// TwinCAT 3 PLC project SILO_OOP_PLC
// ProgramVersion: 3.1.4024.0
// libraries:
//   Tc2_Standard, * (Beckhoff Automation GmbH)
//   Tc2_System, * (Beckhoff Automation GmbH)
//   Tc3_Module, * (Beckhoff Automation GmbH)
// project tree:
//   / PlcTask.TcTTO
//   POUs/1. Interfaces/ itfActuate.TcIO, itfAutoManual.TcIO, itfDetect.TcIO, itfFault.TcIO, itfRamp.TcIO, itfReturnBOOL.TcIO, itfScale.TcIO, itfSiloFlags.TcIO, itfState.TcIO, itfStatusFlags.TcIO
//   POUs/2. Features/ itfActuateImplement.TcPOU, itfFaultImplement.TcPOU, itfRampImplement.TcPOU, itfScaleAnalogInputImplement.TcPOU, itfScaleAnalogOutputImplement.TcPOU, itfDetectImplement.TcPOU, itfSiloFlagsImplement.TcPOU, itfStatusFlagsImplement.TcPOU
//   POUs/3. IO Structure/ GateI.TcDUT, GateO.TcDUT, LoadCellI.TcDUT, LoadCellO.TcDUT, MotorI.TcDUT, MotorO.TcDUT, ProxI.TcDUT, VFDI.TcDUT, VFDO.TcDUT
//   POUs/4. Actuators/ Gate.TcPOU, Motor.TcPOU, VFD.TcPOU
//   POUs/5. Sensors/ LoadCell.TcPOU, ProximitySensor.TcPOU
//   POUs/6.Wrapper/ Wrapper.TcPOU
//   POUs/7.FSM/ BaseState.TcPOU, BufferingProduct.TcPOU, ConveyProduct.TcPOU, Dose.TcPOU, DoseInit.TcPOU, GateHandler.TcPOU, MixerDepositCheck.TcPOU, Mixing.TcPOU, NewBatch.TcPOU, StorageCheck.TcPOU
//   POUs/ MAIN.TcPOU
// real-time tasks:
//   TASK PlcTask: cycle T#10ms, priority 20, ADS port 350

CONFIGURATION SILO_OOP_PLC
    RESOURCE PLC ON TwinCAT3
        TASK PlcTask(INTERVAL := T#10ms, PRIORITY := 20);
        PROGRAM MAIN WITH PlcTask : MAIN;
    END_RESOURCE
END_CONFIGURATION

// ---- POUs/3. IO Structure/GateI.TcDUT
TYPE GateI :
STRUCT
	Open : BOOL;
	Close : BOOL;
END_STRUCT
END_TYPE

// ---- POUs/3. IO Structure/GateO.TcDUT
TYPE GateO :
STRUCT
	Coil : BOOL;
END_STRUCT
END_TYPE

// ---- POUs/3. IO Structure/LoadCellI.TcDUT
TYPE LoadCellI :
STRUCT
	AnalogSignal : INT;
	MaxSignalValue : INT;
	MaxUnitValue : INT;
END_STRUCT
END_TYPE

// ---- POUs/3. IO Structure/LoadCellO.TcDUT
TYPE LoadCellO :
STRUCT
	ScaledValue : INT;
END_STRUCT
END_TYPE

// ---- POUs/3. IO Structure/MotorI.TcDUT
TYPE MotorI :
STRUCT
	Start : BOOL;
	Stop : BOOL;
	Overload : BOOL;
	ResetOverload: BOOL;
END_STRUCT
END_TYPE

// ---- POUs/3. IO Structure/MotorO.TcDUT
TYPE MotorO :
STRUCT
	Coil : BOOL;
	FaultStatus : BOOL;
END_STRUCT
END_TYPE

// ---- POUs/3. IO Structure/ProxI.TcDUT
TYPE ProxI :
STRUCT
	Signal : BOOL;
END_STRUCT
END_TYPE

// ---- POUs/3. IO Structure/VFDI.TcDUT
TYPE VFDI EXTENDS MotorI :
STRUCT
	InputFreq : INT;
	RampRate : INT;
	FreqMaxSignal : INT;
END_STRUCT
END_TYPE

// ---- POUs/3. IO Structure/VFDO.TcDUT
TYPE VFDO EXTENDS MotorO :
STRUCT
	OutputFreq : INT;
END_STRUCT
END_TYPE

// ---- POUs/1. Interfaces/itfActuate.TcIO
INTERFACE itfActuate

METHOD mTurnOffAuto : BOOL
VAR_INPUT
END_VAR
END_METHOD

METHOD mTurnOffManual : BOOL
VAR_INPUT
END_VAR
END_METHOD

METHOD mTurnOnAuto : BOOL
VAR_INPUT
END_VAR
END_METHOD

METHOD mTurnOnManual : BOOL
VAR_INPUT
END_VAR
END_METHOD

PROPERTY pCoil : Bool
GET
END_GET
SET
END_SET
END_PROPERTY

PROPERTY pStart : Bool
GET
END_GET
SET
END_SET
END_PROPERTY

PROPERTY pStop : Bool
GET
END_GET
SET
END_SET
END_PROPERTY

END_INTERFACE

// ---- POUs/1. Interfaces/itfAutoManual.TcIO
INTERFACE itfAutoManual

METHOD mAutoOff : BOOL
VAR_INPUT
END_VAR
END_METHOD

METHOD mAutoOn : BOOL
VAR_INPUT
END_VAR
END_METHOD

METHOD mFault : BOOL
VAR_INPUT
END_VAR
END_METHOD

METHOD mManual : BOOL
VAR_INPUT
END_VAR
END_METHOD

METHOD mRunning : BOOL
VAR_INPUT
END_VAR
END_METHOD

END_INTERFACE

// ---- POUs/1. Interfaces/itfDetect.TcIO
INTERFACE itfDetect

PROPERTY pDetectSignal : BOOL
GET
END_GET
SET
END_SET
END_PROPERTY

END_INTERFACE

// ---- POUs/1. Interfaces/itfFault.TcIO
INTERFACE itfFault

METHOD mResetFault : BOOL
VAR_INPUT
END_VAR
END_METHOD

METHOD mSetFault : BOOL
VAR_INPUT
END_VAR
END_METHOD

PROPERTY pFault : Bool
GET
END_GET
SET
END_SET
END_PROPERTY

PROPERTY pFaultStatus : Bool
GET
END_GET
SET
END_SET
END_PROPERTY

PROPERTY pResetButton : BOOL
GET
END_GET
SET
END_SET
END_PROPERTY

END_INTERFACE

// ---- POUs/1. Interfaces/itfRamp.TcIO
INTERFACE itfRamp

METHOD mDoneTargetFreq : BOOL
VAR_INPUT
END_VAR
END_METHOD

METHOD mRampDown : INT
VAR_INPUT
END_VAR
END_METHOD

METHOD mRampUp : INT
VAR_INPUT
END_VAR
END_METHOD

METHOD mTimerScale : INT
VAR_INPUT
END_VAR
END_METHOD

PROPERTY pOutputValue : INT
GET
END_GET
SET
END_SET
END_PROPERTY

PROPERTY pPulsePeriod : INT
GET
END_GET
SET
END_SET
END_PROPERTY

PROPERTY pRampDone : BOOL
GET
END_GET
SET
END_SET
END_PROPERTY

PROPERTY pRampRate : INT
GET
END_GET
SET
END_SET
END_PROPERTY

PROPERTY pTargetFreq : INT
GET
END_GET
SET
END_SET
END_PROPERTY

END_INTERFACE

// ---- POUs/1. Interfaces/itfReturnBOOL.TcIO
INTERFACE itfReturnBOOL

METHOD mReturnBOOL : BOOL
VAR_INPUT
END_VAR
END_METHOD

END_INTERFACE

// ---- POUs/1. Interfaces/itfScale.TcIO
INTERFACE itfScale

METHOD mScale : INT
VAR_INPUT
END_VAR
END_METHOD

PROPERTY pAnalogSignal : INT
GET
END_GET
SET
END_SET
END_PROPERTY

PROPERTY pMaxSignalValue : INT
GET
END_GET
SET
END_SET
END_PROPERTY

PROPERTY pMaxUnitValue : INT
GET
END_GET
SET
END_SET
END_PROPERTY

PROPERTY pScaledSignal : INT
GET
END_GET
SET
END_SET
END_PROPERTY

END_INTERFACE

// ---- POUs/1. Interfaces/itfSiloFlags.TcIO
INTERFACE itfSiloFlags

PROPERTY pBufferedWeight : INT
GET
END_GET
SET
END_SET
END_PROPERTY

PROPERTY pLowProduct : BOOL
GET
END_GET
SET
END_SET
END_PROPERTY

PROPERTY pTargetWeight : INT
GET
END_GET
SET
END_SET
END_PROPERTY

END_INTERFACE

// ---- POUs/1. Interfaces/itfState.TcIO
INTERFACE itfState

METHOD mIrun : BOOL
VAR_INPUT
END_VAR
END_METHOD

END_INTERFACE

// ---- POUs/1. Interfaces/itfStatusFlags.TcIO
INTERFACE itfStatusFlags

PROPERTY pBuffering : BOOL
GET
END_GET
SET
END_SET
END_PROPERTY

PROPERTY pDosing : BOOL
GET
END_GET
SET
END_SET
END_PROPERTY

PROPERTY pFault : BOOL
GET
END_GET
SET
END_SET
END_PROPERTY

PROPERTY pHaltBatch : BOOL
GET
END_GET
SET
END_SET
END_PROPERTY

PROPERTY pLowProduct : BOOL
GET
END_GET
SET
END_SET
END_PROPERTY

PROPERTY pMixing : BOOL
GET
END_GET
SET
END_SET
END_PROPERTY

PROPERTY pStoring : BOOL
GET
END_GET
SET
END_SET
END_PROPERTY

END_INTERFACE

// ---- POUs/MAIN.TcPOU
PROGRAM MAIN
VAR
	Machine1: Wrapper;
	SpiralInput: ARRAY [1..NUM_SILOS] OF VFDI := [(InputFreq := 50, RampRate := 15, FreqMaxSignal := 200), (InputFreq := 45, RampRate := 20, FreqMaxSignal := 200)];
	LoadCellInput: ARRAY [1..NUM_SILOS] OF LoadCellI := [(AnalogSignal := 4000, MaxSignalValue := 10000, MaxUnitValue := 5000), (AnalogSignal := 3000, MaxSignalValue := 10000, MaxUnitValue := 5000)];
	ConveyorInput: ARRAY [1..NUM_CONVEYORS] OF MotorI;
	ElevatorInput: ARRAY [1..NUM_ELEVATORS] OF MotorI;
	MixerInput: ARRAY [1..NUM_MIXERS] OF VFDI;
	GateInput: ARRAY [1..NUM_GATES] OF GateI;
	ProximityInput: ARRAY [1..NUM_PROXIMITY] OF ProxI;
	SpiralOutput: ARRAY [1..NUM_SILOS] OF VFDO;
	LoadCellOutput: ARRAY [1..NUM_SILOS] OF LoadCellO;
	ConveyorOutput: ARRAY [1..NUM_CONVEYORS] OF MotorO;
	ElevatorOutput: ARRAY [1..NUM_ELEVATORS] OF MotorO;
	MixerOutput: ARRAY [1..NUM_MIXERS] OF VFDO;
	GateOutput: ARRAY [1..NUM_GATES] OF GateO;
	
	Buffering : BOOL;
	Dosing : BOOL;
	Fault : BOOL;
	HaltBatch : BOOL;
	Mixing : BOOL;
	Sorting : BOOL;
	
END_VAR
VAR CONSTANT
	NUM_SILOS : INT:=2;
	NUM_GATES : INT:=2;
	NUM_CONVEYORS : INT:=1;
	NUM_ELEVATORS : INT:=1;
	NUM_PROXIMITY : INT:=4;
	NUM_MIXERS : INT:=1;
END_VAR

Machine1(
	SpiralInput:= SpiralInput , 
	LoadCellInput:= LoadCellInput, 
	ConveyorInput:= ConveyorInput, 
	ElevatorInput:= ElevatorInput, 
	MixerInput:= MixerInput, 
	GateInput:= GateInput, 
	ProximityInput:= ProximityInput, 
	SpiralOutput=> SpiralOutput, 
	LoadCellOutput=> LoadCellOutput, 
	ConveyorOutput=> ConveyorOutput, 
	ElevatorOutput=> ElevatorOutput, 
	MixerOutput=> MixerOutput, 
	GateOutput=> GateOutput);

Machine1.SiloFlagsAccessI[1].pTargetWeight := 50;
Machine1.SiloFlagsAccessI[2].pTargetWeight := 80;
	
Buffering := Machine1.MachineFlagsAccessI.pBuffering;
Dosing := Machine1.MachineFlagsAccessI.pDosing;
Fault := Machine1.MachineFlagsAccessI.pFault;
HaltBatch := Machine1.MachineFlagsAccessI.pHaltBatch;
Mixing := Machine1.MachineFlagsAccessI.pMixing;
Sorting := Machine1.MachineFlagsAccessI.pStoring;

END_PROGRAM

// ---- POUs/6.Wrapper/Wrapper.TcPOU
FUNCTION_BLOCK Wrapper
VAR_INPUT
	SpiralInput : ARRAY [1..NUM_SILOS] OF VFDI;
	LoadCellInput : ARRAY [1..NUM_SILOS] OF LoadCellI;
	ConveyorInput : ARRAY [1..NUM_CONVEYORS] OF MotorI;
	ElevatorInput : ARRAY [1..NUM_ELEVATORS] OF MotorI;
	MixerInput : ARRAY [1..NUM_MIXERS] OF VFDI;
	GateInput : ARRAY [1..NUM_GATES] OF GateI;
	ProximityInput : ARRAY [1..NUM_PROXIMITY] OF ProxI;
	
	SpiralAccessI : ARRAY [1..NUM_SILOS] OF itfAutoManual;
	ConveyorAccessI : ARRAY [1..NUM_CONVEYORS] OF itfAutoManual;
	ElevatorAccessI : ARRAY [1..NUM_ELEVATORS] OF itfAutoManual;
	MixerAccessI : ARRAY [1..NUM_MIXERS] OF itfAutoManual;
	GateAccessI : ARRAY [1..NUM_GATES] OF itfAutoManual;
	ProximityAccessI : ARRAY [1..NUM_PROXIMITY] OF itfReturnBOOL;
	MachineFlagsAccessI : itfStatusFlags;
	SiloFlagsAccessI : ARRAY [1..NUM_SILOS] OF itfSiloFlags;
	
	SuperActuator : ARRAY [1..NUM_ACTUATORS] OF itfAutoManual;	
END_VAR
VAR_OUTPUT
	SpiralOutput : ARRAY [1..NUM_SILOS] OF VFDO;
	LoadCellOutput : ARRAY [1..NUM_SILOS] OF LoadCellO;
	ConveyorOutput : ARRAY [1..NUM_CONVEYORS] OF MotorO;
	ElevatorOutput : ARRAY [1..NUM_ELEVATORS] OF MotorO;
	MixerOutput : ARRAY [1..NUM_MIXERS] OF VFDO;
	GateOutput : ARRAY [1..NUM_GATES] OF GateO;
END_VAR
VAR

////////////////////////////////////Actuators//////////////////////////////////////////
	Spiral : ARRAY [0..NUM_SILOS] OF VFD;
	Conveyor : ARRAY [0..NUM_CONVEYORS] OF Motor;
	Elevator : ARRAY [0..NUM_ELEVATORS] OF Motor;
	Mixer : ARRAY [0..NUM_MIXERS] OF VFD;
	Gate : ARRAY [0..NUM_SILOS] OF Gate;
////////////////////////////////////Sensors////////////////////////////////////////////
	LoadCell : ARRAY [0..NUM_SILOS] OF LoadCell;
	Proximities : ARRAY [0..NUM_PROXIMITY] OF ProximitySensor;
///////////////////////////////Machine Flags///////////////////////////////////////////
	MachineFlags : itfStatusFlagsImplement;	
	SiloFlags : ARRAY [0..NUM_SILOS] OF itfSiloFlagsImplement;
	
	INDEX : INT;
	StateIndex : INT := 1;
	IndependentStateIndex : INT :=1;
//////////////////////////////////FSM///////////////////////////////////////////////////
	Execute : ARRAY [1..NUM_STATES] OF itfState;
	Execute_Independent : ARRAY [1..NUM_INDEPENDENT_STATES] OF itfState;
	
	Buffer : BufferingProduct(THIS);
	Convey : ConveyProduct(THIS);
	DoseInitialize : DoseInit(THIS);
	DoseBegin : Dose(THIS);
	Mix : Mixing (THIS);
	GateActuate : GateHandler(THIS);
	Guard : NewBatch(THIS);
	Store : StorageCheck(THIS);
	MixerCheck : MixerDepositCheck(THIS);
//////////////////////////////Fault Handling//////////////////////////////////////////////
	LastStatus : ARRAY[1..NUM_ACTUATORS] OF BOOL;
	
	FaultR : R_TRIG;
	FaultF : F_TRIG;
	
END_VAR
VAR CONSTANT
	NUM_SILOS : INT:=2;
	NUM_GATES : INT:=2;
	NUM_CONVEYORS : INT:=1;
	NUM_ELEVATORS : INT:=1;
	NUM_PROXIMITY : INT:=4;
	NUM_MIXERS : INT:=1;
	
	NUM_ACTUATORS : INT:=7;
	
	NUM_STATES : INT:=9;
	NUM_INDEPENDENT_STATES : INT:=1;
END_VAR

Map();
mManualMode();
StatesMap();

FaultR(CLK:=mCheckFaults());
FaultF(CLK:=mCheckFaults());

IF FaultR.Q THEN
	mSaveActuatorsStatus();
	mGeneralShutDown();
END_IF

IF FaultF.Q THEN
	mRestoreStatus();
END_IF

IF mCheckFaults()=FALSE THEN
	IF pStateIndex > NUM_STATES THEN
		pStateIndex := 1;
	ELSE
		Execute[pStateIndex].mIrun();
	END_IF
	
	Execute_Independent[pIndependentStateIndex].mIrun();
END_IF

METHOD PRIVATE Map : BOOL
VAR_INPUT
END_VAR
FOR INDEX:=1 TO NUM_SILOS BY 1 DO
	SpiralAccessI[INDEX] := Spiral[INDEX];
	Spiral[INDEX](VFDInput:= SpiralInput[INDEX], VFDOutput=>SpiralOutput[INDEX]);
	
	LoadCell[INDEX](LoadCellInput := LoadCellInput[INDEX], LoadCellOutput => LoadCellOutput[INDEX]);

	SiloFlagsAccessI[INDEX] := SiloFlags[INDEX];
END_FOR

FOR INDEX:=1 TO NUM_CONVEYORS BY 1 DO
	ConveyorAccessI[INDEX] := Conveyor[INDEX];
	Conveyor[INDEX](MotorInput:=ConveyorInput[INDEX], MotorOutput=>ConveyorOutput[INDEX]);
END_FOR

FOR INDEX:=1 TO NUM_ELEVATORS BY 1 DO
	ElevatorAccessI[INDEX] := Elevator[INDEX];
	Elevator[INDEX](MotorInput:=ElevatorInput[INDEX], MotorOutput=>ElevatorOutput[INDEX]);
END_FOR

FOR INDEX:=1 TO NUM_MIXERS BY 1 DO
	MixerAccessI[INDEX] := Mixer[INDEX];
	Mixer[INDEX](VFDInput:=MixerInput[INDEX], VFDOutput=>MixerOutput[INDEX]);
END_FOR

FOR INDEX:=1 TO NUM_GATES BY 1 DO
	Gate[INDEX](GateInput:=GateInput[INDEX], GateOutput=>GateOutput[INDEX]);
	GateAccessI[INDEX] := Gate[INDEX];
END_FOR

FOR INDEX:=1 TO NUM_PROXIMITY BY 1 DO
	Proximities[INDEX](ProximityInput:=ProximityInput[INDEX]);
	ProximityAccessI[INDEX] := Proximities[INDEX];
END_FOR

MachineFlagsAccessI := MachineFlags;

SuperActuator[1] := SpiralAccessI[1];
SuperActuator[2] := SpiralAccessI[2];
SuperActuator[3] := ConveyorAccessI[1];
SuperActuator[4] := ElevatorAccessI[1];
SuperActuator[5] := MixerAccessI[1];
SuperActuator[6] := GateAccessI[1];
SuperActuator[7] := GateAccessI[2];
END_METHOD

METHOD PRIVATE mCheckFaults : BOOL
VAR_INPUT
END_VAR
FOR INDEX:=1 TO NUM_ACTUATORS BY 1 DO
	IF SuperActuator[INDEX].mFault() THEN
	THIS^.MachineFlagsAccessI.pFault:=TRUE;
	mCheckFaults:=TRUE;
	RETURN;
END_IF	
END_FOR

MachineFlagsAccessI.pFault:=FALSE;
mCheckFaults:=FALSE;
END_METHOD

METHOD PRIVATE mGeneralShutDown : BOOL
VAR_INPUT
END_VAR
FOR INDEX:=1 TO NUM_ACTUATORS BY 1 DO
	SuperActuator[INDEX].mAutoOff();
END_FOR
END_METHOD

METHOD PRIVATE mManualMode : BOOL
VAR_INPUT
END_VAR
FOR INDEX:=1 TO NUM_ACTUATORS BY 1 DO
	SuperActuator[INDEX].mManual();	
END_FOR
END_METHOD

METHOD PRIVATE mRestoreStatus : BOOL
VAR_INPUT
END_VAR
FOR INDEX:=1 TO NUM_ACTUATORS BY 1 DO
	IF LastStatus[INDEX] = TRUE THEN
		SuperActuator[INDEX].mAutoOn();
	END_IF
END_FOR
END_METHOD

METHOD PRIVATE mSaveActuatorsStatus : BOOL
VAR_INPUT
END_VAR
FOR INDEX:=1 TO NUM_ACTUATORS BY 1 DO
	LastStatus[INDEX]:=SuperActuator[INDEX].mRunning();
END_FOR
END_METHOD

PROPERTY pIndependentStateIndex : INT
GET
pIndependentStateIndex := IndependentStateIndex;
END_GET
SET
IndependentStateIndex := pIndependentStateIndex;
END_SET
END_PROPERTY

PROPERTY pNUM_SILOS : INT
GET
pNUM_SILOS := NUM_SILOS;
END_GET
END_PROPERTY

PROPERTY pStateIndex : INT
GET
pStateIndex := StateIndex;
END_GET
SET
StateIndex := pStateIndex;
END_SET
END_PROPERTY

METHOD PRIVATE StatesMap : BOOL
VAR_INPUT
END_VAR
Execute[1]:=Guard;
Execute[2]:=Convey;
Execute[3]:=DoseInitialize;
Execute[4]:=DoseBegin;
Execute[5]:=Buffer;
Execute[6]:=MixerCheck;
Execute[7]:=GateActuate;
Execute[8]:=Mix;
Execute[9]:=GateActuate;

Execute_Independent[1]:=Store;

CASE pStateIndex OF
	4:
	Buffer.mStateInit(BufferingTime:=T#8S);
	5:
	GateActuate.mStateInit(GateTime:=T#10S, GateNumber:=1);
	6:
	Mix.mStateInit(MixingTime:=T#15S);
	7:
	GateActuate.mStateInit(GateTime:=T#15S, GateNumber:=2);
END_CASE
END_METHOD

END_FUNCTION_BLOCK

// ---- POUs/4. Actuators/VFD.TcPOU
FUNCTION_BLOCK VFD IMPLEMENTS itfAutoManual
VAR_INPUT
	VFDInput : VFDI;
END_VAR
VAR_OUTPUT
	VFDOutput : VFDO;
END_VAR
VAR
	MotorComp : Motor;
	MotorIref : REFERENCE TO MotorI;
	MotorOref : REFERENCE TO MotorO;

	ScaleComp : itfScaleAnalogOutputImplement;
	Scale : itfScale;

	RampComp : itfRampImplement;
	Ramp : itfRamp;
	
	CoilR : R_TRIG;
	CoilF : F_TRIG;
	
	FlagUp : BOOL;
	FlagDown : BOOL;
END_VAR

Map();

CoilR(CLK:= MotorOref.Coil);
CoilF(CLK:= MotorOref.Coil);

METHOD PRIVATE Map : BOOL
VAR_INPUT
END_VAR
MotorIref REF= VFDInput;
MotorOref REF= VFDOutput;
MotorComp(MotorInput := MotorIref, MotorOutput => MotorOref);

Scale := ScaleComp;
Ramp := RampComp;

Ramp.pTargetFreq := VFDInput.InputFreq;
Ramp.pRampRate := VFDInput.RampRate;

Scale.pMaxSignalValue := VFDInput.FreqMaxSignal;
Scale.pAnalogSignal := Ramp.pOutputValue;
VFDOutput.OutputFreq := Scale.pScaledSignal;
Scale.mScale();
END_METHOD

{warning 'add method implementation '}
METHOD mAutoOff : BOOL
RampFreq();
MotorComp.mAutoOff();
END_METHOD

{warning 'add method implementation '}
METHOD mAutoOn : BOOL
RampFreq();
MotorComp.mAutoOn();
END_METHOD

{warning 'add method implementation '}
METHOD mFault : BOOL
mFault := MotorComp.mFault();
END_METHOD

{warning 'add method implementation '}
METHOD mManual : BOOL
RampFreq();
MotorComp.mManual();
END_METHOD

{warning 'add method implementation '}
METHOD mRunning : BOOL
mRunning := MotorComp.mRunning();
END_METHOD

METHOD RampFreq : INT
VAR_INPUT
END_VAR
IF CoilR.Q THEN
	FlagUp := TRUE;
	// Setting Flag
	FlagDown := FALSE;
END_IF

IF CoilF.Q THEN
	FlagDown := TRUE;
	// Setting Flag
	FlagUp := FALSE;
END_IF

IF FlagUp THEN
	//FlagDown := FALSE;
	Ramp.mRampUp();
	IF Ramp.pRampDone THEN
		FlagUp := FALSE;
	END_IF
END_IF

IF FlagDown THEN
	//FlagUp := FALSE;
	Ramp.mRampDown();
	IF Ramp.pOutputValue = 0 THEN
		FlagDown := FALSE;
	END_IF
END_IF
END_METHOD

END_FUNCTION_BLOCK

// ---- POUs/4. Actuators/Motor.TcPOU
FUNCTION_BLOCK Motor IMPLEMENTS itfAutoManual
VAR_INPUT
	MotorInput : MotorI;
END_VAR
VAR_OUTPUT
	MotorOutput : MotorO;
END_VAR
VAR
	Actuate : itfActuate;
	Fault : itfFault;
	
	ActuateComp : itfActuateImplement;
	FaultComp : itfFaultImplement;
END_VAR

Map();
FaultHandler();

METHOD PROTECTED FaultHandler : BOOL
VAR_INPUT
END_VAR
Fault.mResetFault();
Fault.mSetFault();
END_METHOD

METHOD PRIVATE Map : BOOL
VAR_INPUT
END_VAR
Actuate := ActuateComp;
Fault := FaultComp;

Actuate.pStart := MotorInput.Start;
Actuate.pStop := MotorInput.Stop;
MotorOutput.Coil := Actuate.pCoil;
MotorOutput.FaultStatus := Fault.pFaultStatus;

Fault.pResetButton := MotorInput.ResetOverload;
Fault.pFault := MotorInput.Overload;
END_METHOD

{warning 'add method implementation '}
METHOD mAutoOff : BOOL
Actuate.mTurnOffAuto();
END_METHOD

{warning 'add method implementation '}
METHOD mAutoOn : BOOL
IF mFault() = FALSE THEN
Actuate.mTurnOnAuto();
END_IF
END_METHOD

{warning 'add method implementation '}
METHOD mFault : BOOL
mFault := Fault.pFaultStatus;
END_METHOD

{warning 'add method implementation '}
METHOD mManual : BOOL
IF mFault() = FALSE THEN
Actuate.mTurnOnManual();
END_IF
Actuate.mTurnOffManual();
END_METHOD

{warning 'add method implementation '}
METHOD mRunning : BOOL
mRunning := Actuate.pCoil;
END_METHOD

END_FUNCTION_BLOCK

// ---- POUs/2. Features/itfActuateImplement.TcPOU
FUNCTION_BLOCK itfActuateImplement IMPLEMENTS itfActuate
VAR_INPUT
END_VAR
VAR_OUTPUT
END_VAR
VAR
	Coil : BOOL;
	Start : BOOL;
	Stop : BOOL;
END_VAR

METHOD mTurnOffAuto : BOOL
pCoil := FALSE;
END_METHOD

METHOD mTurnOffManual : BOOL
IF pStop THEN
	pCoil := FALSE;
END_IF
END_METHOD

METHOD mTurnOnAuto : BOOL
pCoil := TRUE;
END_METHOD

METHOD mTurnOnManual : BOOL
IF pStart THEN
	pCoil := TRUE;
END_IF
END_METHOD

{warning 'add property implementation'}
PROPERTY pCoil : BOOL
GET
pCoil := Coil;
END_GET
SET
Coil := pCoil;
END_SET
END_PROPERTY

{warning 'add property implementation'}
PROPERTY pStart : BOOL
GET
pStart := Start;
END_GET
SET
Start := pStart;
END_SET
END_PROPERTY

{warning 'add property implementation'}
PROPERTY pStop : BOOL
GET
pStop := Stop;
END_GET
SET
Stop := pStop;
END_SET
END_PROPERTY

END_FUNCTION_BLOCK

// ---- POUs/2. Features/itfFaultImplement.TcPOU
FUNCTION_BLOCK itfFaultImplement IMPLEMENTS itfFault
VAR_INPUT
END_VAR
VAR_OUTPUT
END_VAR
VAR
	Fault : BOOL;
	FaultStatus : BOOL;
	ResetButton : BOOL;
END_VAR

METHOD mResetFault : BOOL
IF pResetButton AND NOT pFault THEN
	pFaultStatus := FALSE;
END_IF
END_METHOD

METHOD mSetFault : BOOL
IF pFault THEN
	pFaultStatus := TRUE;
	mSetFault := TRUE;
END_IF
END_METHOD

{warning 'add property implementation'}
PROPERTY pFault : BOOL
GET
pFault := Fault;
END_GET
SET
Fault := pFault;
END_SET
END_PROPERTY

{warning 'add property implementation'}
PROPERTY pFaultStatus : BOOL
GET
pFaultStatus := FaultStatus;
END_GET
SET
FaultStatus := pFaultStatus;
END_SET
END_PROPERTY

{warning 'add property implementation'}
PROPERTY pResetButton : BOOL
GET
pResetButton := ResetButton;
END_GET
SET
ResetButton := pResetButton;
END_SET
END_PROPERTY

END_FUNCTION_BLOCK

// ---- POUs/2. Features/itfScaleAnalogOutputImplement.TcPOU
FUNCTION_BLOCK itfScaleAnalogOutputImplement EXTENDS itfScaleAnalogInputImplement
VAR_INPUT
END_VAR
VAR_OUTPUT
END_VAR
VAR
END_VAR

METHOD mScale : INT
pScaledSignal := pAnalogSignal * pMaxSignalValue;
END_METHOD

END_FUNCTION_BLOCK

// ---- POUs/2. Features/itfScaleAnalogInputImplement.TcPOU
FUNCTION_BLOCK itfScaleAnalogInputImplement IMPLEMENTS itfScale
VAR_INPUT
END_VAR
VAR_OUTPUT
END_VAR
VAR
	AnalogSignal : INT;
	MaxSignalValue : INT;
	MaxUnitValue : INT;
	ScaledSignal : INT;
END_VAR

METHOD mScale : INT
pScaledSignal := pAnalogSignal * pMaxUnitValue / pMaxSignalValue;
END_METHOD

{warning 'add property implementation'}
PROPERTY pAnalogSignal : INT
GET
pAnalogSignal := AnalogSignal;
END_GET
SET
AnalogSignal := pAnalogSignal;
END_SET
END_PROPERTY

{warning 'add property implementation'}
PROPERTY pMaxSignalValue : INT
GET
IF MaxSignalValue > 0 THEN
pMaxSignalValue := MaxSignalValue;
ELSE
	pMaxSignalValue := 1;
END_IF
END_GET
SET
MaxSignalValue := pMaxSignalValue;
END_SET
END_PROPERTY

{warning 'add property implementation'}
PROPERTY pMaxUnitValue : INT
GET
pMaxUnitValue := MaxUnitValue;
END_GET
SET
MaxUnitValue := pMaxUnitValue;
END_SET
END_PROPERTY

{warning 'add property implementation'}
PROPERTY pScaledSignal : INT
GET
pScaledSignal := ScaledSignal;
END_GET
SET
ScaledSignal := pScaledSignal;
END_SET
END_PROPERTY

END_FUNCTION_BLOCK

// ---- POUs/2. Features/itfRampImplement.TcPOU
FUNCTION_BLOCK itfRampImplement IMPLEMENTS itfRamp
VAR_INPUT
END_VAR
VAR_OUTPUT
END_VAR
VAR
	OutputValue : INT;
	RampDone : BOOL;
	RampRate : INT;
	TargetFreq : INT;
	PulsePeriod : INT;
	Timer : TON;
END_VAR

METHOD mDoneTargetFreq : BOOL
IF pOutputValue >= pTargetFreq THEN
	pRampDone := TRUE;
	ELSE
		pRampDone := FALSE;
END_IF
END_METHOD

METHOD mRampDown : INT
mTimerScale();
mDoneTargetFreq();

IF TIMER.Q THEN
	IF pOutputValue > 0 THEN
pOutputValue := pOutputValue - 1;
	END_IF
END_IF
END_METHOD

METHOD mRampUp : INT
mTimerScale();
mDoneTargetFreq();

IF TIMER.Q THEN
	IF pOutputValue < pTargetFreq THEN
pOutputValue := pOutputValue + 1;
	END_IF
END_IF
END_METHOD

METHOD mTimerScale : INT
pPulsePeriod := (pRampRate * 1000) / TargetFreq;

TIMER(IN:= NOT TIMER.Q, PT:= INT_TO_TIME(pPulsePeriod));
END_METHOD

PROPERTY pOutputValue : INT
GET
pOutputValue := OutputValue;
END_GET
SET
OutputValue := pOutputValue;
END_SET
END_PROPERTY

PROPERTY pPulsePeriod : INT
GET
pPulsePeriod := PulsePeriod;
END_GET
SET
PulsePeriod := pPulsePeriod;
END_SET
END_PROPERTY

PROPERTY pRampDone : BOOL
GET
pRampDone := RampDone;
END_GET
SET
RampDone := pRampDone;
END_SET
END_PROPERTY

PROPERTY pRampRate : INT
GET
pRampRate := RampRate;
END_GET
SET
RampRate := pRampRate;
END_SET
END_PROPERTY

PROPERTY pTargetFreq : INT
GET
IF TargetFreq > 0 THEN
pTargetFreq := TargetFreq;
ELSE
	pTargetFreq := 1;
END_IF
END_GET
SET
VAR
	END_IFTargetFreq: INT;
END_VAR
IF pTargetFreq > 0 THEN
TargetFreq := pTargetFreq;
ELSE
	TargetFreq := 1;
END_IF
END_SET
END_PROPERTY

END_FUNCTION_BLOCK

// ---- POUs/4. Actuators/Gate.TcPOU
FUNCTION_BLOCK Gate Implements itfAutoManual
VAR_INPUT
	GateInput : GateI;
END_VAR
VAR_OUTPUT
	GateOutput : GateO;
END_VAR
VAR
Actuate : itfActuate;
ActuateComp : itfActuateImplement;	

END_VAR

Map();

METHOD PRIVATE Map : BOOL
VAR_INPUT
END_VAR
Actuate := ActuateComp;

Actuate.pStart := GateInput.Open;
Actuate.pStop := GateInput.Close;
GateOutput.Coil := Actuate.pCoil;
END_METHOD

{warning 'add method implementation '}
METHOD mAutoOff : BOOL
Actuate.mTurnOffAuto();
END_METHOD

{warning 'add method implementation '}
METHOD mAutoOn : BOOL
Actuate.mTurnOnAuto();
END_METHOD

{warning 'add method implementation '}
METHOD mFault : BOOL
END_METHOD

{warning 'add method implementation '}
METHOD mManual : BOOL
Actuate.mTurnOnManual();
Actuate.mTurnOffManual();
END_METHOD

{warning 'add method implementation '}
METHOD mRunning : BOOL
mRunning := Actuate.pCoil;
END_METHOD

END_FUNCTION_BLOCK

// ---- POUs/5. Sensors/LoadCell.TcPOU
FUNCTION_BLOCK LoadCell
VAR_INPUT
	LoadCellInput : LoadCellI;
END_VAR
VAR_OUTPUT
	LoadCellOutput : LoadCellO;
END_VAR
VAR
	ScaleComp : itfScaleAnalogInputImplement;
	Scale : itfScale;
END_VAR

Map();
Scale.mScale();

METHOD PRIVATE Map : BOOL
VAR_INPUT
END_VAR
Scale := ScaleComp;
Scale.pAnalogSignal := LoadCellInput.AnalogSignal;
Scale.pMaxSignalValue := LoadCellInput.MaxSignalValue;
Scale.pMaxUnitValue := LoadCellInput.MaxUnitValue;

LoadCellOutput.ScaledValue :=Scale.pScaledSignal;
END_METHOD

END_FUNCTION_BLOCK

// ---- POUs/5. Sensors/ProximitySensor.TcPOU
FUNCTION_BLOCK ProximitySensor IMPLEMENTS itfReturnBOOL
VAR_INPUT
	ProximityInput : ProxI;
END_VAR
VAR_OUTPUT
END_VAR
VAR
	ProxComp : itfDetectImplement;
	Prox : itfDetect;
END_VAR

Map();

METHOD PRIVATE Map : BOOL
VAR_INPUT
END_VAR
Prox := ProxComp;
Prox.pDetectSignal := ProximityInput.Signal;
END_METHOD

{warning 'add method implementation '}
METHOD mReturnBOOL : BOOL
mReturnBOOL := Prox.pDetectSignal;
END_METHOD

END_FUNCTION_BLOCK

// ---- POUs/2. Features/itfDetectImplement.TcPOU
FUNCTION_BLOCK itfDetectImplement IMPLEMENTS itfDetect
VAR_INPUT
END_VAR
VAR_OUTPUT
END_VAR
VAR
	DetectSignal : BOOL;
END_VAR

{warning 'add property implementation'}
PROPERTY pDetectSignal : BOOL
GET
pDetectSignal := DetectSignal;
END_GET
SET
DetectSignal := pDetectSignal;
END_SET
END_PROPERTY

END_FUNCTION_BLOCK

// ---- POUs/2. Features/itfStatusFlagsImplement.TcPOU
FUNCTION_BLOCK itfStatusFlagsImplement IMPLEMENTS itfStatusFlags
VAR_INPUT
END_VAR
VAR_OUTPUT
END_VAR
VAR
	Buffering : BOOL;
	Dosing : BOOL;
	Fault : BOOL;
	HaltBatch : BOOL;
	Mixing : BOOL;
	Storing : BOOL;
	LowProduct : BOOL;
END_VAR

{warning 'add property implementation'}
PROPERTY pBuffering : BOOL
GET
pBuffering := Buffering;
END_GET
SET
Buffering := pBuffering;
END_SET
END_PROPERTY

{warning 'add property implementation'}
PROPERTY pDosing : BOOL
GET
pDosing := Dosing;
END_GET
SET
Dosing := pDosing;
END_SET
END_PROPERTY

{warning 'add property implementation'}
PROPERTY pFault : BOOL
GET
pFault := Fault;
END_GET
SET
Fault := pFault;
END_SET
END_PROPERTY

{warning 'add property implementation'}
PROPERTY pHaltBatch : BOOL
GET
pHaltBatch := HaltBatch;
END_GET
SET
HaltBatch := pHaltBatch;
END_SET
END_PROPERTY

{warning 'add property implementation'}
PROPERTY pLowProduct : BOOL
GET
pLowProduct := LowProduct;
END_GET
SET
LowProduct := pLowProduct;
END_SET
END_PROPERTY

{warning 'add property implementation'}
PROPERTY pMixing : BOOL
GET
pMixing := Mixing;
END_GET
SET
Mixing := pMixing;
END_SET
END_PROPERTY

{warning 'add property implementation'}
PROPERTY pStoring : BOOL
GET
pStoring := Storing;
END_GET
SET
Storing := pStoring;
END_SET
END_PROPERTY

END_FUNCTION_BLOCK

// ---- POUs/7.FSM/Mixing.TcPOU
FUNCTION_BLOCK Mixing EXTENDS BaseState
VAR_INPUT
END_VAR
VAR_OUTPUT
END_VAR
VAR
	InternalMixingTime : TIME;
END_VAR

METHOD mIrun : BOOL
StateTimer(IN:=TRUE, PT:=InternalMixingTime);
BasePointer^.MachineFlagsAccessI.pMixing := TRUE;
IF StateTimer.Q THEN
	mNextState();
	BasePointer^.MachineFlagsAccessI.pMixing := FALSE;
	StateTimer(IN:=FALSE);
END_IF
END_METHOD

METHOD mStateInit : BOOL
VAR_INPUT
	MixingTime : TIME;
END_VAR
InternalMixingTime := MixingTime;
END_METHOD

END_FUNCTION_BLOCK

// ---- POUs/7.FSM/BaseState.TcPOU
FUNCTION_BLOCK BaseState IMPLEMENTS itfState
VAR_INPUT
	BasePointer : POINTER TO WRAPPER;
END_VAR
VAR_OUTPUT
END_VAR
VAR
	StateTimer : TON;
	Index : INT;
	TESTING : INT;
END_VAR

METHOD FB_INIT : BOOL
VAR_INPUT
	bInitRetains : BOOL;
	bInCopyCode : BOOL;
	WrapperPointer : POINTER TO Wrapper;
END_VAR
BasePointer := WrapperPointer;
END_METHOD

METHOD PROTECTED mCheckDosing : BOOL
VAR_INPUT
END_VAR
FOR INDEX :=1 TO BasePointer^.pNUM_SILOS BY 1 DO
	IF BasePointer^.SpiralAccessI[INDEX].mRunning() THEN
		RETURN;
	END_IF
END_FOR

mCheckDosing := TRUE;
END_METHOD

METHOD mIrun : BOOL
END_METHOD

METHOD mNextState : BOOL
VAR_INPUT
END_VAR
StateTimer(IN:= TRUE, PT:= T#1000MS);

IF StateTimer.Q THEN
BasePointer^.pStateIndex := BasePointer^.pStateIndex + 1;
StateTimer(IN:= FALSE);
END_IF
END_METHOD

END_FUNCTION_BLOCK

// ---- POUs/2. Features/itfSiloFlagsImplement.TcPOU
FUNCTION_BLOCK itfSiloFlagsImplement IMPLEMENTS itfSiloFlags
VAR_INPUT
END_VAR
VAR_OUTPUT
END_VAR
VAR
	BufferedWeight : INT;
	TargetWeight : INT;
	LowProduct : BOOL;
END_VAR

PROPERTY pBufferedWeight : INT
GET
pBufferedWeight := BufferedWeight;
END_GET
SET
BufferedWeight := pBufferedWeight;
END_SET
END_PROPERTY

PROPERTY pLowProduct : BOOL
GET
pLowProduct := LowProduct;
END_GET
SET
LowProduct := pLowProduct;
END_SET
END_PROPERTY

PROPERTY pTargetWeight : INT
GET
pTargetWeight := TargetWeight;
END_GET
SET
TargetWeight := pTargetWeight;
END_SET
END_PROPERTY

END_FUNCTION_BLOCK

// ---- POUs/7.FSM/BufferingProduct.TcPOU
FUNCTION_BLOCK BufferingProduct EXTENDS BaseState
VAR_INPUT
END_VAR
VAR_OUTPUT
END_VAR
VAR
	InternalBufferingTime : TIME;
END_VAR

METHOD mIrun : BOOL
IF BasePointer^.ProximityAccessI[1].mReturnBOOL() THEN;
	IF mCheckDosing() THEN
		StateTimer(IN:= TRUE, PT:=InternalBufferingTime);
		IF StateTimer.Q = TRUE THEN
			mNextState();
			StateTimer(IN:= FALSE);
//		ELSE
//			RETURN;
		END_IF
	END_IF
END_IF
END_METHOD

METHOD mStateInit : BOOL
VAR_INPUT
	BufferingTime : TIME;
END_VAR
InternalBufferingTime := BufferingTime;
END_METHOD

END_FUNCTION_BLOCK

// ---- POUs/7.FSM/ConveyProduct.TcPOU
FUNCTION_BLOCK ConveyProduct EXTENDS BaseState
VAR_INPUT
END_VAR
VAR_OUTPUT
END_VAR
VAR
END_VAR

METHOD mIrun : BOOL
BasePointer^.ConveyorAccessI[1].mAutoOn();
BasePointer^.ElevatorAccessI[1].mAutoOn();
BasePointer^.MixerAccessI[1].mAutoOn();
mNextState();
END_METHOD

END_FUNCTION_BLOCK

// ---- POUs/7.FSM/DoseInit.TcPOU
FUNCTION_BLOCK DoseInit EXTENDS BaseState
VAR_INPUT
END_VAR
VAR_OUTPUT
END_VAR
VAR
END_VAR

METHOD mIrun : BOOL
FOR Index:=1 TO BasePointer^.pNUM_SILOS BY 1 DO
	IF BasePointer^.LoadCellOutput[INDEX].ScaledValue < BasePointer^.SiloFlagsAccessI[INDEX].pTargetWeight THEN
		BasePointer^.SiloFlagsAccessI[INDEX].pLowProduct := TRUE;	
	ELSE
		BasePointer^.SiloFlagsAccessI[INDEX].pLowProduct := FALSE;
	END_IF
		
	BasePointer^.SiloFlagsAccessI[Index].pBufferedWeight := BasePointer^.LoadCellOutput[Index].ScaledValue;
	BasePointer^.SpiralAccessI[Index].mAutoOn();
	BasePointer^.MachineFlagsAccessI.pDosing := TRUE;
END_FOR

mNextState();
END_METHOD

END_FUNCTION_BLOCK

// ---- POUs/7.FSM/Dose.TcPOU
FUNCTION_BLOCK Dose EXTENDS BaseState
VAR_INPUT
END_VAR
VAR_OUTPUT
END_VAR
VAR
END_VAR

METHOD mIrun : BOOL
FOR INDEX:=1 TO BasePointer^.pNUM_SILOS BY 1 DO
	IF BasePointer^.SiloFlagsAccessI[INDEX].pBufferedWeight - BasePointer^.LoadCellOutput[INDEX].ScaledValue >= BasePointer^.SiloFlagsAccessI[INDEX].pTargetWeight THEN
		BasePointer^.SpiralAccessI[INDEX].mAutoOff();
	END_IF
END_FOR

IF mCheckDosing() = TRUE THEN
	BasePointer^.MachineFlagsAccessI.pDosing := FALSE;
	ELSE
		RETURN;
END_IF

mNextState();
END_METHOD

END_FUNCTION_BLOCK

// ---- POUs/7.FSM/GateHandler.TcPOU
FUNCTION_BLOCK GateHandler EXTENDS BaseState
VAR_INPUT
END_VAR
VAR_OUTPUT
END_VAR
VAR
	InternalGateTime : TIME;
	InternalGateNumber : INT;
END_VAR

METHOD mIrun : BOOL
BasePointer^.GateAccessI[InternalGateNumber].mAutoOn();
StateTimer(IN:= TRUE, PT:=InternalGateTime);
IF StateTimer.Q THEN
	BasePointer^.GateAccessI[InternalGateNumber].mAutoOff();
	mNextState();
	StateTimer(IN:= FALSE);
END_IF
END_METHOD

METHOD mStateInit : BOOL
VAR_INPUT
	GateTime : TIME;
	GateNumber : INT;
END_VAR
InternalGateTime := GateTime;
InternalGateNumber := GateNumber;
END_METHOD

END_FUNCTION_BLOCK

// ---- POUs/7.FSM/NewBatch.TcPOU
FUNCTION_BLOCK NewBatch EXTENDS BaseState
VAR_INPUT
END_VAR
VAR_OUTPUT
END_VAR
VAR
END_VAR

METHOD mIrun : BOOL
IF BasePointer^.MachineFlagsAccessI.pBuffering = TRUE THEN
	BasePointer^.MachineFlagsAccessI.pHaltBatch := TRUE;
ELSE
	BasePointer^.MachineFlagsAccessI.pHaltBatch := FALSE;
	mNextState();	
END_IF
END_METHOD

END_FUNCTION_BLOCK

// ---- POUs/7.FSM/StorageCheck.TcPOU
FUNCTION_BLOCK StorageCheck EXTENDS BaseState
VAR_INPUT
END_VAR
VAR_OUTPUT
END_VAR
VAR
END_VAR

METHOD mIrun : BOOL
IF BasePointer^.ProximityAccessI[1].mReturnBOOL() THEN
	BasePointer^.MachineFlagsAccessI.pBuffering := TRUE;
	ELSE
		BasePointer^.MachineFlagsAccessI.pBuffering := FALSE;
END_IF

IF BasePointer^.ProximityAccessI[2].mReturnBOOL() THEN
	BasePointer^.MachineFlagsAccessI.pStoring := TRUE;
	ELSE
		BasePointer^.MachineFlagsAccessI.pStoring := FALSE;
END_IF

FOR INDEX:=1 TO BasePointer^.pNUM_SILOS BY 1 DO
	IF BasePointer^.SiloFlagsAccessI[INDEX].pLowProduct THEN
		BasePointer^.MachineFlagsAccessI.pLowProduct:=TRUE;
		EXIT;
	END_IF
	TESTING := 5;
END_FOR
END_METHOD

END_FUNCTION_BLOCK

// ---- POUs/7.FSM/MixerDepositCheck.TcPOU
FUNCTION_BLOCK MixerDepositCheck EXTENDS BaseState
VAR_INPUT
END_VAR
VAR_OUTPUT
END_VAR
VAR
END_VAR

METHOD mIrun : BOOL
IF BasePointer^.MachineFlagsAccessI.pStoring THEN
	RETURN;
ELSE
		mNextState();
END_IF
END_METHOD

END_FUNCTION_BLOCK
